TYPE ST_DIS_Chanel_Diagnosis :
STRUCT
	bWirebreak 				: BOOL;
	bPowerSupplymissing	: BOOL;
END_STRUCT
END_TYPE

(* stored: Version 1.1.0.1
   DUT ST_DIS_Chanel_Diagnosis: Id {242ceead-e935-4bf0-a04e-e57f7c8bd04c} *)
